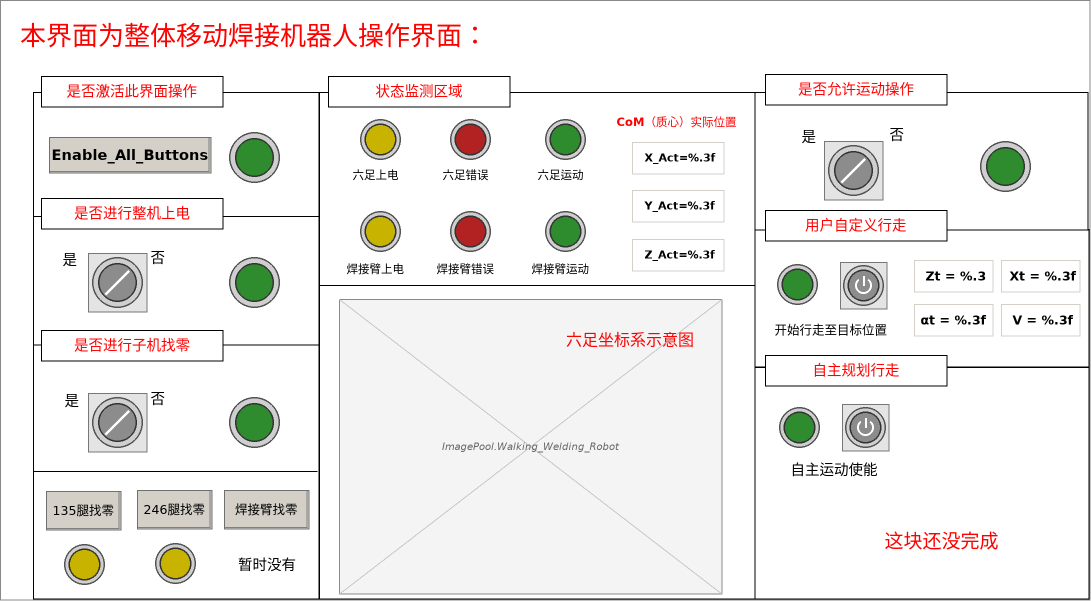
VISUALIZATION Visu_Walking_Welding_Robot_Control  // 1091x601
    Rectangle (754,367 335x232)
    Rectangle (754,229 335x138)
    Rectangle (753,92 335x138)
    Rectangle (33,92 286x125)
    Rectangle (319,92 436x194)
    Rectangle (319,285 436x314)
    Rectangle (33,344 286x255)
    Label (17,15 583x42), "本界面为整体移动焊接机器人操作界面："
    Rectangle (33,216 286x129)
    Lamp1 (225,252 59x61), variable: Walking_Welding_Robot_Control.Walking_Welding_Robot_Power, style: Lamp-Lamp1-Green
    RotarySwitch (88,252 59x61), variable: Walking_Welding_Robot_Control.Walking_Welding_Robot_Power, behaviour: TOGGLE, style: Switch-RotarySwitch-Gray
    Label (138,243 40x30), "否"
    Label (50,245 40x30), "是"
    Rectangle (41,198 182x31), "是否进行整机上电"
    Lamp1 (355,116 51x47), variable: Walking_Robot_Control.Robot_Power, style: Lamp-Lamp1-Yellow
    Lamp1 (445,116 51x47), variable: Walking_Robot_Control.Robot_Error, style: Lamp-Lamp1-Red
    Label (422,159 87x32), "六足错误"
    Label (332,159 87x32), "六足上电"
    Lamp1 (445,208 51x47), variable: Welding_Arm_Control.Robot_Error, style: Lamp-Lamp1-Red
    Label (422,253 87x32), "焊接臂错误"
    Lamp1 (355,208 51x47), variable: Welding_Arm_Control.Robot_Power, style: Lamp-Lamp1-Yellow
    Label (332,253 87x32), "焊接臂上电"
    RotarySwitch (88,392 59x61), variable: Walking_Welding_Robot_Control.Walking_Welding_Robot_Home_Execute, behaviour: TOGGLE, style: Switch-RotarySwitch-Gray
    Rectangle (41,330 182x31), "是否进行子机找零"
    Lamp1 (225,392 59x61), variable: Walking_Welding_Robot_Control.Walking_Welding_Robot_Home_Execute, style: Lamp-Lamp1-Green
    Label (138,384 40x30), "否"
    Label (52,386 40x30), "是"
    Rectangle (765,74 182x31), "是否允许运动操作"
    Lamp1 (976,136 59x61), variable: Walking_Welding_Robot_Control.Walking_Welding_Robot_Moving_Execute, style: Lamp-Lamp1-Green
    Button (137,490 75x39), "246腿找零"
        tap Walking_Robot_Control.Leg_Home_Set[2]
    Button (46,491 75x39), "135腿找零"
        tap Walking_Robot_Control.Leg_Home_Set[1]
    Button (224,490 85x39), "焊接臂找零"
        tap Welding_Arm_Control.Welding_Arm_Home_Set
    Lamp1 (59,541 51x47), variable: Walking_Robot_Control.Tripod_Home_Done[1], style: Lamp-Lamp1-Yellow
    Lamp1 (150,540 51x47), variable: Walking_Robot_Control.Tripod_Home_Done[2], style: Lamp-Lamp1-Yellow
    Rectangle (765,210 182x31), "用户自定义行走"
    Textfield (914,260 79x32), "Zt = %.3", text variable: Walking_Welding_Robot_Control.Robot_Walking_Z
        OnMouseClick: write Robot_Movement.t_IntervalWalking_Welding_Robot_Control.Robot_Walking_ZWalking_Welding_Robot_Control.Robot_Walking_Z via Default
    Textfield (1001,260 79x32), "Xt = %.3f", text variable: Walking_Welding_Robot_Control.Robot_Walking_X
        OnMouseClick: write Robot_Movement.t_IntervalWalking_Welding_Robot_Control.Robot_Walking_XWalking_Welding_Robot_Control.Robot_Walking_X via Default
    Textfield (914,304 79x32), "αt = %.3f", text variable: Walking_Welding_Robot_Control.Robot_Walking_alpha
        OnMouseClick: write Robot_Movement.t_IntervalWalking_Welding_Robot_Control.Robot_Walking_alphaWalking_Welding_Robot_Control.Robot_Walking_alpha via Default
    Textfield (1001,304 79x32), "V = %.3f", text variable: Walking_Welding_Robot_Control.Robot_Walking_Velocity
        OnMouseClick: write Robot_Movement.t_IntervalWalking_Welding_Robot_Control.Robot_Walking_VelocityWalking_Welding_Robot_Control.Robot_Walking_Velocity via Default
    Lamp1 (772,261 51x47), variable: Walking_Welding_Robot_Control.User_Moving_Control, style: Lamp-Lamp1-Green
    PowerSwitch (838,262 51x47), variable: Walking_Welding_Robot_Control.User_Moving_Control, behaviour: TOGGLE, style: Switch-PowerSwitch-Gray
    Image (339,299 383x295), image: ImagePool.Walking_Welding_Robot
    Textfield (632,239 92x32), "Z_Act=%.3f", text variable: Walking_Robot_Movement.Act_Slice[3]
    Textfield (632,142 92x32), "X_Act=%.3f", text variable: Walking_Robot_Movement.Act_Slice[4]
    Textfield (632,190 92x32), "Y_Act=%.3f", text variable: Walking_Robot_Movement.Act_Slice[5]
    Lamp1 (540,116 51x47), variable: Walking_Robot_Movement.ExtSetPointEnable, style: Lamp-Lamp1-Green
    Lamp1 (540,208 51x47), variable: Welding_Arm_Movement.ExtSetPointEnable, style: Lamp-Lamp1-Green
    Label (517,159 87x32), "六足运动"
    Label (517,253 87x32), "焊接臂运动"
    Rectangle (765,355 182x31), "自主规划行走"
    PowerSwitch (840,404 51x47), variable: Walking_Welding_Robot_Control.Auto_Moving_Control, behaviour: TOGGLE, style: Switch-PowerSwitch-Gray
    Lamp1 (774,404 51x47), variable: Walking_Welding_Robot_Control.Auto_Moving_Control, style: Lamp-Lamp1-Green
    Label (781,454 106x32), "自主运动使能"
    Button (49,137 162x36), "Enable_All_Buttons"
        toggle Walking_Welding_Robot_Control.Walking_Welding_Robot_Joint_Control
    Lamp1 (225,127 59x61), variable: Walking_Welding_Robot_Control.Walking_Welding_Robot_Joint_Control, style: Lamp-Lamp1-Green
    Label (759,314 144x32), "开始行走至目标位置"
    Line (33,471) (317,471)
    Rectangle (328,76 182x31), "状态监测区域"
    Rectangle (41,76 182x31), "是否激活此界面操作"
    Label (526,325 208x30), "六足坐标系示意图"
    Label (603,107 147x30), "CoM（质心）实际位置"
    Label (223,549 88x32), "暂时没有"
    Label (877,120 40x30), "否"
    Label (789,122 40x30), "是"
    RotarySwitch (824,140 59x61), variable: Walking_Welding_Robot_Control.Walking_Welding_Robot_Moving_Execute, behaviour: TOGGLE, style: Switch-RotarySwitch-Gray
    Label (851,525 181x32), "这块还没完成"
END_VISUALIZATION

(* stored: Version 1.1.0.1, ProductVersion 3.1.4020.12
   Visu Visu_Walking_Welding_Robot_Control: Id {29749d12-5fcc-4a58-ab75-42edc3f0ea40} *)
